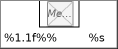
VISUALIZATION VISU_VANNE_ASS_H  // 118x49
VAR_IN_OUT
	m_Input_VANNE : BLOCK_VVAT_650_NO;
END_VAR

VAR_INPUT
	m_Input_NumFrame_Manu:	USINT;		(*numéro de frame à afficher dans le synoptique MANUEL*)
END_VAR
    Rectangle (0,0 118x49), invisible if: TRUE
    Polygon (0,0), colour toggle: m_Input_VANNE.STATE_Lam
    Rectangle (76,28 41x20), "%s", text variable: m_Input_VANNE.MNEMO
    Polygon (0,0), colour toggle: m_Input_VANNE.STATE_On, invisible if: NOT (m_Input_VANNE.STATE_Off OR m_Input_VANNE.STATE_On)
    Ellipse (54,2 10x10), colour toggle: m_Input_VANNE.STATE_Ok, invisible if: NOT m_Input_VANNE.STATE_Ok
    Rectangle (1,28 77x20), "%1.1f%%", text variable: m_Input_VANNE.STATE_Position
    Image (47,1 26x25), invisible if: NOT m_Input_VANNE.STATE_Nok, image: MesImages.warning
    Rectangle (39,0 40x27), invisible if: NOT m_Input_VANNE.MANUAL
        OnMouseClick: execute { .VISU_INDEX_MANU := m_Input_NumFrame_Manu; }
        OnMouseClick: change screen: SYN_MANUEL
END_VISUALIZATION

(* stored: Version 1.1.0.1, ProductVersion 3.1.4026.18
   Visu VISU_VANNE_ASS_H: Id {6ec437b0-429e-4617-8d0e-2db7fa570a26} *)
